Fanuc KAREL source: IO0190.KL

PROGRAM IO0190
%STACKSIZE=65535
%PRIORITY=65535
%NOLOCKGROUP
ROUTINE RTEST FROM IO0190
ROUTINE RTEST
VAR
L1 : ARRAY[3] OF INTEGER
L2 : XYZWPR
L3 : JOINTPOS9
L4 : POSITION
U2C_37 : INTEGER
U2C_38 : REAL
U2C_39 : REAL
U2C_40 : BOOLEAN
U2C_41 : REAL
BEGIN
U2C_37=1
L1[1]=2
U2C_40=TRUE
U2C_41=1.0
-- UNRESOLVED_PC line 19 opcodes [27 27 9D 19 2E 29 64 29 6C 76 21 1A] marker_code=77
END RTEST
BEGIN
RTEST
END IO0190
